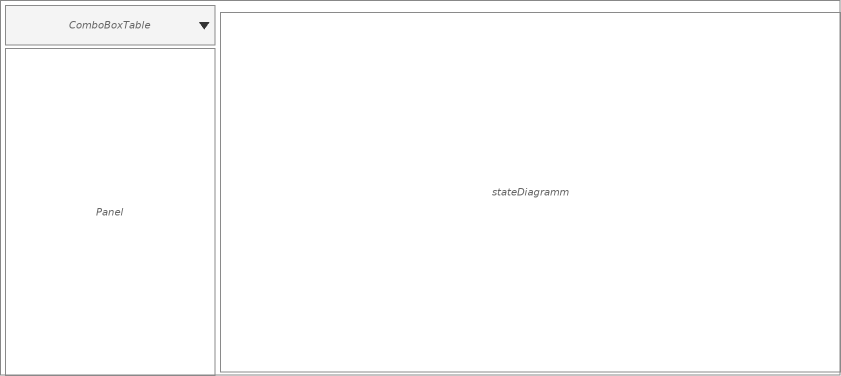
VISUALIZATION Visualization  // 841x376
    ComboBoxTable (5,5 210x40), variable: MAIN.Visualisierung.VisuSelectedZustandsautomat, data array: MAIN.Visualisierung.VisuNamenZustandsautomaten
        p3854506369: MAIN.Visualisierung.VisuNamenZustandsautomaten[INDEX]
    Frame (5,48 210x328)
        shows Panel(Panel := MAIN.Visualisierung.VisuPanel)
    Frame (220,12 621x360)
        shows stateDiagramm(Panel := MAIN.Visualisierung.VisuPanel)
END_VISUALIZATION

(* stored: Version 1.1.0.1, ProductVersion 3.1.4024.9
   Visu Visualization: Id {061e6f26-a4a7-436c-a180-de9e666e4536} *)
